(* PLC project syrup, Dassault Systèmes ControlBuild 2024x *)
(* stored: creationDateTime 2023-10-03T11:13:39-01:00 *)

FUNCTION_BLOCK faults
  VAR_INPUT
    generalFault1 : BOOL := false;
    generalFault2 : BOOL := false;
    generalFault3 : BOOL := false;
    generalFault4 : BOOL := false;
  END_VAR
  VAR_OUTPUT
    fault : BOOL := false;
  END_VAR

(* LD diagram, written out as Structured Text *)
1:
fault := generalFault4 OR generalFault1 OR generalFault2 OR generalFault3;
END_FUNCTION_BLOCK

PROGRAM batch.syrup
  VAR_INPUT
    syrup1Weight : DINT := 0;
    syrup2Weight : DINT := 0;
    syrup3Weight : DINT := 0;
  END_VAR
  VAR_INPUT
    cycleInProgress : BOOL := false;
    weighingRequest : BOOL := false;
    acknowledgePB : BOOL := false;
  END_VAR
  VAR_INPUT
    autoMode : BOOL := false;
    manualMode : BOOL := false;
  END_VAR
  VAR_OUTPUT
    weighingOk : BOOL := false;
    fault : BOOL := false;
    syrupExtraction : REAL := 0.0;
  END_VAR

(* FBD diagram, written out as Structured Text *)
arrivalValveSyrup1(acknowledgePB := acknowledgePB, autoMode := autoMode, manualMode := manualMode, autoCloseCmd := syrupManagement.introS1End, autoOpenCmd := syrupManagement.introduceS1);
arrivalValveSyrup2(acknowledgePB := acknowledgePB, autoMode := autoMode, manualMode := manualMode, autoCloseCmd := syrupManagement.introS2End, autoOpenCmd := syrupManagement.introduceS2);
arrivalValveSyrup3(acknowledgePB := acknowledgePB, autoMode := autoMode, manualMode := manualMode, autoCloseCmd := syrupManagement.introS3End, autoOpenCmd := syrupManagement.introduceS3);
syrupQuantity(flowSyrup1 := arrivalValveSyrup1.outputFlow, flowSyrup2 := arrivalValveSyrup2.outputFlow, flowSyrup3 := arrivalValveSyrup3.outputFlow);
flow(inputFlow := syrupsTank.tankLevel);
syrupExtractionValve(acknowledgePB := acknowledgePB, autoMode := autoMode, manualMode := manualMode, autoCloseCmd := syrupManagement.exitSyrupEnd, autoOpenCmd := syrupManagement.exitSyrup, inputFlow := flow.outputFlow);
syrupsTank(inletFlow := syrupQuantity.flow, outletFlow := syrupExtractionValve.outputFlow);
level(measure := syrupsTank.tankLevel);
scale(inputValue := level.realValue);
syrupManagement(weighingRequest := weighingRequest, cycleInProgress := cycleInProgress, weighingWeight := scale.dintValue, syrup1Weight := syrup1Weight, syrup2Weight := syrup2Weight, syrup3Weight := syrup3Weight);
weighingOk := syrupManagement.weighingOk;
faults1(generalFault1 := arrivalValveSyrup1.generalFault, generalFault2 := arrivalValveSyrup2.generalFault, generalFault3 := arrivalValveSyrup3.generalFault, generalFault4 := syrupExtractionValve.generalFault);
fault := faults1.fault;
syrupExtraction := syrupExtractionValve.outputFlow;
END_PROGRAM
